# EPICS autosave request: soft_iocs/meas_comp_e1608/iocBoot/iocmeas_comp_e1608/auto_settings.req
file "E1608_settings.req", P=18ID:E1608:
